FUNCTION_BLOCK FB_Module01 EXTENDS FB_Component
VAR_INPUT
END_VAR
VAR_OUTPUT
END_VAR
VAR
	fbLogger:					FB_LoggerFactory;
	fbTcLogger:					FB_TcLogger;
	fbAlarm:					FB_Alarm;
	fbComponent1:				FB_Component;
	fbComponent2:				FB_Component;
	fbComponent3:				FB_Component;
	fbComponent4:				FB_ComponentEX;
	nIndex:						INT;
	fbComponent:				ARRAY[1..1000] OF FB_Component;
END_VAR

METHOD PUBLIC M_Attach
VAR_INPUT
	Component:		I_Component;
END_VAR
Component.P_Event.P_Logger:= fbLogger;
Component.P_Observer.M_Attach(THIS^);
fbObserver.M_Attach(Component);
END_METHOD

METHOD PUBLIC M_Cycle
VAR_INPUT
END_VAR
SUPER^.M_Cycle();

fbComponent1.M_Cycle();
fbComponent2.M_Cycle();
fbComponent3.M_Cycle();
fbComponent4.M_Cycle();

FOR nIndex:= 1 TO 1000 DO 
	fbComponent[nIndex].M_Cycle();
END_FOR;
END_METHOD

METHOD PUBLIC M_Dettach
VAR_INPUT
	Component:		I_Component;
END_VAR
Component.P_Event.P_Logger:= 0;
Component.P_Observer.M_Detach(THIS^);
fbObserver.M_Detach(Component);
END_METHOD

METHOD PROTECTED M_Initialise : BOOL
VAR_INPUT
END_VAR
IF SUPER^.M_Initialise() THEN
	fbEvent.P_Logger:= fbLogger;
	fbLogger.M_Add(fbAlarm);
	fbLogger.M_Add(fbTcLogger);

	M_Attach(fbComponent1);
	M_Attach(fbComponent2);
	M_Attach(fbComponent3);
	M_Attach(fbComponent4);
	
	
	FOR nIndex:= 1 TO 1000 DO 
		M_Attach(fbComponent[nIndex]);
	END_FOR;
	
	
	
	M_Initialise:= TRUE;
END_IF
END_METHOD

METHOD PROTECTED M_Resetting : BOOL
VAR_INPUT
END_VAR
VAR
	nIndex:					DINT;
END_VAR
M_Resetting:= TRUE;
WHILE nIndex < fbObserver.nLength DO
	fbObserver.M_Index(nIndex).M_Request(E_Request.Reset);
	nIndex:= nIndex +1;
END_WHILE

fbAlarm.M_Reset();
END_METHOD

METHOD PROTECTED M_Running
VAR_INPUT
END_VAR
IF NOT M001.fbPowerOn.P_Value THEN
	fbEvent.M_Add(M001.fbPowerOn.P_ID);
	fbEvent.M_Error('Power not on', 2 ,E_Behaviour.Abort);
ELSIF NOT M001.fbFuse1.P_Value THEN
	fbEvent.M_Add(M001.fbFuse1.P_ID);
	fbEvent.M_Error('Fuse Triped', 3 ,E_Behaviour.Stop);	
	
END_IF

fbEvent.M_Warning('My first Warning', 4 );
END_METHOD

METHOD PROTECTED M_Starting : BOOL
VAR_INPUT
END_VAR
VAR
	nIndex:					DINT;
END_VAR
M_Starting:= TRUE;
WHILE nIndex < fbObserver.nLength DO
	M_Starting:= M_Starting AND fbObserver.M_Index(nIndex).M_Request(E_Request.Start);
	nIndex:= nIndex +1;
END_WHILE
END_METHOD

END_FUNCTION_BLOCK

(* stored: Version 1.1.0.1, ProductVersion 3.1.4024.12
   POU FB_Module01: Id {3744d03d-359c-4ab8-84fb-4ea93b7a5162}, SpecialFunc None
   Method M_Attach: Id {ed0f0a5a-a1be-4f63-bf1a-cd6def284ca3}
   Method M_Cycle: Id {655447dc-389e-494a-be91-78d8a111b7aa}
   Method M_Dettach: Id {01833449-7b04-429a-a301-4e20def83f01}
   Method M_Initialise: Id {714c485c-83a6-4af2-a706-fec3f6b598e5}
   Method M_Resetting: Id {fa00b107-60e3-427f-9569-a0a34888482b}
   Method M_Running: Id {eaffebca-5ff2-4f17-be84-3310a9ace22e}
   Method M_Starting: Id {12752945-7cd6-464f-965a-f81c0b828bfd} *)
